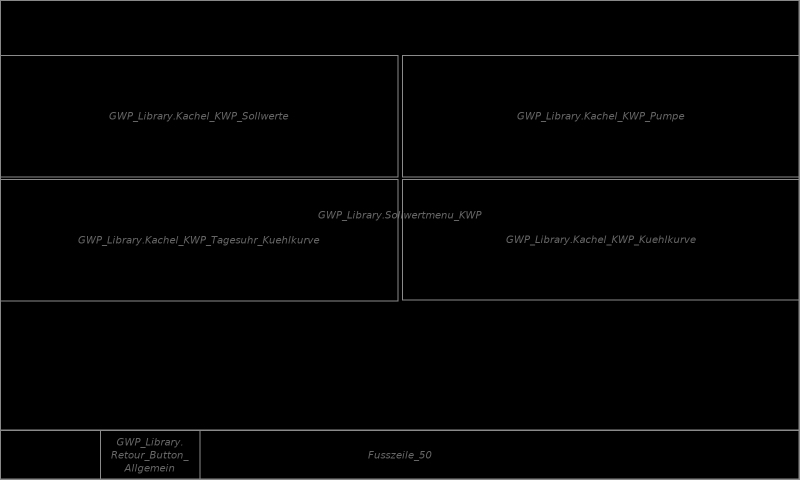
VISUALIZATION Sollwertmenu_KWP  // 800x480
    Frame (0,0 800x430)
        shows GWP_Library.Sollwertmenu_KWP()
    Frame (0,55 398x122)
        shows GWP_Library.Kachel_KWP_Sollwerte(FB_Kreis_3KO := Main.Kreis_3KO_0)
        OnMouseClick: change screen: KWP_SP_AC_NC_Sollwerte
    Frame (402,55 398x122)
        shows GWP_Library.Kachel_KWP_Pumpe()
        OnMouseClick: change screen: KWP_SP_AC_NC_PU_Sollwerte
    Frame (0,179 398x122)
        shows GWP_Library.Kachel_KWP_Tagesuhr_Kuehlkurve()
        OnMouseClick: change screen: KWP_SP_AC_NC_CLK_D
    Frame (402,179 398x121)
        shows GWP_Library.Kachel_KWP_Kuehlkurve()
        OnMouseClick: change screen: KWP_SP_AC_NC_GR_4_ohne_RE
    Frame (0,430 800x50)
        shows Fusszeile_50()
    Frame (100,430 100x50)
        shows GWP_Library.Retour_Button_Allgemein()
END_VISUALIZATION

(* stored: Version 1.1.0.1, ProductVersion 3.1.4022.6
   Visu Sollwertmenu_KWP: Id {5858d207-30f6-4fa6-89d1-c84cb70aab69} *)
